// TIA Portal V20 export
// export: Created 2026-08-08T00:00:00.0000000Z, ExportSetting WithDefaults, DisplayName Totally Integrated Automation Portal, DisplayVersion V20, DisplayName TIA Portal Openness, DisplayVersion V20, DisplayName TIA Portal Version Control Interface, DisplayVersion V20, DisplayName STEP 7 Professional, DisplayVersion V20, DisplayName STEP 7 Safety, DisplayVersion V20, DisplayName WinCC Basic/Comfort/Advanced, DisplayVersion V20, DisplayName WinCC Professional, DisplayVersion V20, DisplayName WinCC Unified, DisplayVersion V20
FUNCTION "FC_PhysicalIoCopy" : Void   // FC, SCL
{ S7_Optimized_Access := 'TRUE' }
VERSION : 0.1
// NOT YET WIRED INTO Main[OB1]. Generated 2026-08-08 from the real addresses confirmed live in TIA's Device overview after assigning all 3 ET200SP stations (AFT/MID/FWD) to PLC_1's PROFINET IO system - before that, every module showed no address at all. This is the only block in the whole project that references real physical %I/%Q addresses; everything downstream (FC_IoMapper, Valve_Channels_DB) only ever deals with the abstract 1..368 / 1..208 channel numbers in IO_Buffer_DB. Still needs: (1) FB_ValveLoop simulation guard for real-mapped valves, (2) both this and FC_IoMapper actually called from Main[OB1] - see FC_IoMapper's own header comment. Safe to have present unwired: it only touches IO_Buffer_DB, which nothing else reads yet.
// stored: AutoNumber true, IsIECCheckEnabled false, SetENOAutomatically false, UDAEnableTagReadback false
BEGIN
// Network 1

       // === DIGITAL INPUTS: real %I bits -> IO_Buffer_DB.DI[1..368] ===
       // -- AFT DI modules --
       "IO_Buffer_DB".DI[1] := %I2.0;
       "IO_Buffer_DB".DI[2] := %I2.1;
       "IO_Buffer_DB".DI[3] := %I2.2;
       "IO_Buffer_DB".DI[4] := %I2.3;
       "IO_Buffer_DB".DI[5] := %I2.4;
       "IO_Buffer_DB".DI[6] := %I2.5;
       "IO_Buffer_DB".DI[7] := %I2.6;
       "IO_Buffer_DB".DI[8] := %I2.7;
       "IO_Buffer_DB".DI[9] := %I3.0;
       "IO_Buffer_DB".DI[10] := %I3.1;
       "IO_Buffer_DB".DI[11] := %I3.2;
       "IO_Buffer_DB".DI[12] := %I3.3;
       "IO_Buffer_DB".DI[13] := %I3.4;
       "IO_Buffer_DB".DI[14] := %I3.5;
       "IO_Buffer_DB".DI[15] := %I3.6;
       "IO_Buffer_DB".DI[16] := %I3.7;
       "IO_Buffer_DB".DI[17] := %I4.0;
       "IO_Buffer_DB".DI[18] := %I4.1;
       "IO_Buffer_DB".DI[19] := %I4.2;
       "IO_Buffer_DB".DI[20] := %I4.3;
       "IO_Buffer_DB".DI[21] := %I4.4;
       "IO_Buffer_DB".DI[22] := %I4.5;
       "IO_Buffer_DB".DI[23] := %I4.6;
       "IO_Buffer_DB".DI[24] := %I4.7;
       "IO_Buffer_DB".DI[25] := %I5.0;
       "IO_Buffer_DB".DI[26] := %I5.1;
       "IO_Buffer_DB".DI[27] := %I5.2;
       "IO_Buffer_DB".DI[28] := %I5.3;
       "IO_Buffer_DB".DI[29] := %I5.4;
       "IO_Buffer_DB".DI[30] := %I5.5;
       "IO_Buffer_DB".DI[31] := %I5.6;
       "IO_Buffer_DB".DI[32] := %I5.7;
       "IO_Buffer_DB".DI[33] := %I6.0;
       "IO_Buffer_DB".DI[34] := %I6.1;
       "IO_Buffer_DB".DI[35] := %I6.2;
       "IO_Buffer_DB".DI[36] := %I6.3;
       "IO_Buffer_DB".DI[37] := %I6.4;
       "IO_Buffer_DB".DI[38] := %I6.5;
       "IO_Buffer_DB".DI[39] := %I6.6;
       "IO_Buffer_DB".DI[40] := %I6.7;
       "IO_Buffer_DB".DI[41] := %I7.0;
       "IO_Buffer_DB".DI[42] := %I7.1;
       "IO_Buffer_DB".DI[43] := %I7.2;
       "IO_Buffer_DB".DI[44] := %I7.3;
       "IO_Buffer_DB".DI[45] := %I7.4;
       "IO_Buffer_DB".DI[46] := %I7.5;
       "IO_Buffer_DB".DI[47] := %I7.6;
       "IO_Buffer_DB".DI[48] := %I7.7;
       "IO_Buffer_DB".DI[49] := %I8.0;
       "IO_Buffer_DB".DI[50] := %I8.1;
       "IO_Buffer_DB".DI[51] := %I8.2;
       "IO_Buffer_DB".DI[52] := %I8.3;
       "IO_Buffer_DB".DI[53] := %I8.4;
       "IO_Buffer_DB".DI[54] := %I8.5;
       "IO_Buffer_DB".DI[55] := %I8.6;
       "IO_Buffer_DB".DI[56] := %I8.7;
       "IO_Buffer_DB".DI[57] := %I9.0;
       "IO_Buffer_DB".DI[58] := %I9.1;
       "IO_Buffer_DB".DI[59] := %I9.2;
       "IO_Buffer_DB".DI[60] := %I9.3;
       "IO_Buffer_DB".DI[61] := %I9.4;
       "IO_Buffer_DB".DI[62] := %I9.5;
       "IO_Buffer_DB".DI[63] := %I9.6;
       "IO_Buffer_DB".DI[64] := %I9.7;
       "IO_Buffer_DB".DI[65] := %I10.0;
       "IO_Buffer_DB".DI[66] := %I10.1;
       "IO_Buffer_DB".DI[67] := %I10.2;
       "IO_Buffer_DB".DI[68] := %I10.3;
       "IO_Buffer_DB".DI[69] := %I10.4;
       "IO_Buffer_DB".DI[70] := %I10.5;
       "IO_Buffer_DB".DI[71] := %I10.6;
       "IO_Buffer_DB".DI[72] := %I10.7;
       "IO_Buffer_DB".DI[73] := %I11.0;
       "IO_Buffer_DB".DI[74] := %I11.1;
       "IO_Buffer_DB".DI[75] := %I11.2;
       "IO_Buffer_DB".DI[76] := %I11.3;
       "IO_Buffer_DB".DI[77] := %I11.4;
       "IO_Buffer_DB".DI[78] := %I11.5;
       "IO_Buffer_DB".DI[79] := %I11.6;
       "IO_Buffer_DB".DI[80] := %I11.7;
       "IO_Buffer_DB".DI[81] := %I12.0;
       "IO_Buffer_DB".DI[82] := %I12.1;
       "IO_Buffer_DB".DI[83] := %I12.2;
       "IO_Buffer_DB".DI[84] := %I12.3;
       "IO_Buffer_DB".DI[85] := %I12.4;
       "IO_Buffer_DB".DI[86] := %I12.5;
       "IO_Buffer_DB".DI[87] := %I12.6;
       "IO_Buffer_DB".DI[88] := %I12.7;
       "IO_Buffer_DB".DI[89] := %I13.0;
       "IO_Buffer_DB".DI[90] := %I13.1;
       "IO_Buffer_DB".DI[91] := %I13.2;
       "IO_Buffer_DB".DI[92] := %I13.3;
       "IO_Buffer_DB".DI[93] := %I13.4;
       "IO_Buffer_DB".DI[94] := %I13.5;
       "IO_Buffer_DB".DI[95] := %I13.6;
       "IO_Buffer_DB".DI[96] := %I13.7;
       "IO_Buffer_DB".DI[97] := %I14.0;
       "IO_Buffer_DB".DI[98] := %I14.1;
       "IO_Buffer_DB".DI[99] := %I14.2;
       "IO_Buffer_DB".DI[100] := %I14.3;
       "IO_Buffer_DB".DI[101] := %I14.4;
       "IO_Buffer_DB".DI[102] := %I14.5;
       "IO_Buffer_DB".DI[103] := %I14.6;
       "IO_Buffer_DB".DI[104] := %I14.7;
       "IO_Buffer_DB".DI[105] := %I15.0;
       "IO_Buffer_DB".DI[106] := %I15.1;
       "IO_Buffer_DB".DI[107] := %I15.2;
       "IO_Buffer_DB".DI[108] := %I15.3;
       "IO_Buffer_DB".DI[109] := %I15.4;
       "IO_Buffer_DB".DI[110] := %I15.5;
       "IO_Buffer_DB".DI[111] := %I15.6;
       "IO_Buffer_DB".DI[112] := %I15.7;
       // -- MID DI modules --
       "IO_Buffer_DB".DI[113] := %I16.0;
       "IO_Buffer_DB".DI[114] := %I16.1;
       "IO_Buffer_DB".DI[115] := %I16.2;
       "IO_Buffer_DB".DI[116] := %I16.3;
       "IO_Buffer_DB".DI[117] := %I16.4;
       "IO_Buffer_DB".DI[118] := %I16.5;
       "IO_Buffer_DB".DI[119] := %I16.6;
       "IO_Buffer_DB".DI[120] := %I16.7;
       "IO_Buffer_DB".DI[121] := %I17.0;
       "IO_Buffer_DB".DI[122] := %I17.1;
       "IO_Buffer_DB".DI[123] := %I17.2;
       "IO_Buffer_DB".DI[124] := %I17.3;
       "IO_Buffer_DB".DI[125] := %I17.4;
       "IO_Buffer_DB".DI[126] := %I17.5;
       "IO_Buffer_DB".DI[127] := %I17.6;
       "IO_Buffer_DB".DI[128] := %I17.7;
       "IO_Buffer_DB".DI[129] := %I18.0;
       "IO_Buffer_DB".DI[130] := %I18.1;
       "IO_Buffer_DB".DI[131] := %I18.2;
       "IO_Buffer_DB".DI[132] := %I18.3;
       "IO_Buffer_DB".DI[133] := %I18.4;
       "IO_Buffer_DB".DI[134] := %I18.5;
       "IO_Buffer_DB".DI[135] := %I18.6;
       "IO_Buffer_DB".DI[136] := %I18.7;
       "IO_Buffer_DB".DI[137] := %I19.0;
       "IO_Buffer_DB".DI[138] := %I19.1;
       "IO_Buffer_DB".DI[139] := %I19.2;
       "IO_Buffer_DB".DI[140] := %I19.3;
       "IO_Buffer_DB".DI[141] := %I19.4;
       "IO_Buffer_DB".DI[142] := %I19.5;
       "IO_Buffer_DB".DI[143] := %I19.6;
       "IO_Buffer_DB".DI[144] := %I19.7;
       "IO_Buffer_DB".DI[145] := %I20.0;
       "IO_Buffer_DB".DI[146] := %I20.1;
       "IO_Buffer_DB".DI[147] := %I20.2;
       "IO_Buffer_DB".DI[148] := %I20.3;
       "IO_Buffer_DB".DI[149] := %I20.4;
       "IO_Buffer_DB".DI[150] := %I20.5;
       "IO_Buffer_DB".DI[151] := %I20.6;
       "IO_Buffer_DB".DI[152] := %I20.7;
       "IO_Buffer_DB".DI[153] := %I21.0;
       "IO_Buffer_DB".DI[154] := %I21.1;
       "IO_Buffer_DB".DI[155] := %I21.2;
       "IO_Buffer_DB".DI[156] := %I21.3;
       "IO_Buffer_DB".DI[157] := %I21.4;
       "IO_Buffer_DB".DI[158] := %I21.5;
       "IO_Buffer_DB".DI[159] := %I21.6;
       "IO_Buffer_DB".DI[160] := %I21.7;
       "IO_Buffer_DB".DI[161] := %I22.0;
       "IO_Buffer_DB".DI[162] := %I22.1;
       "IO_Buffer_DB".DI[163] := %I22.2;
       "IO_Buffer_DB".DI[164] := %I22.3;
       "IO_Buffer_DB".DI[165] := %I22.4;
       "IO_Buffer_DB".DI[166] := %I22.5;
       "IO_Buffer_DB".DI[167] := %I22.6;
       "IO_Buffer_DB".DI[168] := %I22.7;
       "IO_Buffer_DB".DI[169] := %I23.0;
       "IO_Buffer_DB".DI[170] := %I23.1;
       "IO_Buffer_DB".DI[171] := %I23.2;
       "IO_Buffer_DB".DI[172] := %I23.3;
       "IO_Buffer_DB".DI[173] := %I23.4;
       "IO_Buffer_DB".DI[174] := %I23.5;
       "IO_Buffer_DB".DI[175] := %I23.6;
       "IO_Buffer_DB".DI[176] := %I23.7;
       "IO_Buffer_DB".DI[177] := %I24.0;
       "IO_Buffer_DB".DI[178] := %I24.1;
       "IO_Buffer_DB".DI[179] := %I24.2;
       "IO_Buffer_DB".DI[180] := %I24.3;
       "IO_Buffer_DB".DI[181] := %I24.4;
       "IO_Buffer_DB".DI[182] := %I24.5;
       "IO_Buffer_DB".DI[183] := %I24.6;
       "IO_Buffer_DB".DI[184] := %I24.7;
       "IO_Buffer_DB".DI[185] := %I25.0;
       "IO_Buffer_DB".DI[186] := %I25.1;
       "IO_Buffer_DB".DI[187] := %I25.2;
       "IO_Buffer_DB".DI[188] := %I25.3;
       "IO_Buffer_DB".DI[189] := %I25.4;
       "IO_Buffer_DB".DI[190] := %I25.5;
       "IO_Buffer_DB".DI[191] := %I25.6;
       "IO_Buffer_DB".DI[192] := %I25.7;
       "IO_Buffer_DB".DI[193] := %I26.0;
       "IO_Buffer_DB".DI[194] := %I26.1;
       "IO_Buffer_DB".DI[195] := %I26.2;
       "IO_Buffer_DB".DI[196] := %I26.3;
       "IO_Buffer_DB".DI[197] := %I26.4;
       "IO_Buffer_DB".DI[198] := %I26.5;
       "IO_Buffer_DB".DI[199] := %I26.6;
       "IO_Buffer_DB".DI[200] := %I26.7;
       "IO_Buffer_DB".DI[201] := %I27.0;
       "IO_Buffer_DB".DI[202] := %I27.1;
       "IO_Buffer_DB".DI[203] := %I27.2;
       "IO_Buffer_DB".DI[204] := %I27.3;
       "IO_Buffer_DB".DI[205] := %I27.4;
       "IO_Buffer_DB".DI[206] := %I27.5;
       "IO_Buffer_DB".DI[207] := %I27.6;
       "IO_Buffer_DB".DI[208] := %I27.7;
       "IO_Buffer_DB".DI[209] := %I28.0;
       "IO_Buffer_DB".DI[210] := %I28.1;
       "IO_Buffer_DB".DI[211] := %I28.2;
       "IO_Buffer_DB".DI[212] := %I28.3;
       "IO_Buffer_DB".DI[213] := %I28.4;
       "IO_Buffer_DB".DI[214] := %I28.5;
       "IO_Buffer_DB".DI[215] := %I28.6;
       "IO_Buffer_DB".DI[216] := %I28.7;
       "IO_Buffer_DB".DI[217] := %I29.0;
       "IO_Buffer_DB".DI[218] := %I29.1;
       "IO_Buffer_DB".DI[219] := %I29.2;
       "IO_Buffer_DB".DI[220] := %I29.3;
       "IO_Buffer_DB".DI[221] := %I29.4;
       "IO_Buffer_DB".DI[222] := %I29.5;
       "IO_Buffer_DB".DI[223] := %I29.6;
       "IO_Buffer_DB".DI[224] := %I29.7;
       // -- FWD DI modules --
       "IO_Buffer_DB".DI[225] := %I30.0;
       "IO_Buffer_DB".DI[226] := %I30.1;
       "IO_Buffer_DB".DI[227] := %I30.2;
       "IO_Buffer_DB".DI[228] := %I30.3;
       "IO_Buffer_DB".DI[229] := %I30.4;
       "IO_Buffer_DB".DI[230] := %I30.5;
       "IO_Buffer_DB".DI[231] := %I30.6;
       "IO_Buffer_DB".DI[232] := %I30.7;
       "IO_Buffer_DB".DI[233] := %I31.0;
       "IO_Buffer_DB".DI[234] := %I31.1;
       "IO_Buffer_DB".DI[235] := %I31.2;
       "IO_Buffer_DB".DI[236] := %I31.3;
       "IO_Buffer_DB".DI[237] := %I31.4;
       "IO_Buffer_DB".DI[238] := %I31.5;
       "IO_Buffer_DB".DI[239] := %I31.6;
       "IO_Buffer_DB".DI[240] := %I31.7;
       "IO_Buffer_DB".DI[241] := %I32.0;
       "IO_Buffer_DB".DI[242] := %I32.1;
       "IO_Buffer_DB".DI[243] := %I32.2;
       "IO_Buffer_DB".DI[244] := %I32.3;
       "IO_Buffer_DB".DI[245] := %I32.4;
       "IO_Buffer_DB".DI[246] := %I32.5;
       "IO_Buffer_DB".DI[247] := %I32.6;
       "IO_Buffer_DB".DI[248] := %I32.7;
       "IO_Buffer_DB".DI[249] := %I33.0;
       "IO_Buffer_DB".DI[250] := %I33.1;
       "IO_Buffer_DB".DI[251] := %I33.2;
       "IO_Buffer_DB".DI[252] := %I33.3;
       "IO_Buffer_DB".DI[253] := %I33.4;
       "IO_Buffer_DB".DI[254] := %I33.5;
       "IO_Buffer_DB".DI[255] := %I33.6;
       "IO_Buffer_DB".DI[256] := %I33.7;
       "IO_Buffer_DB".DI[257] := %I34.0;
       "IO_Buffer_DB".DI[258] := %I34.1;
       "IO_Buffer_DB".DI[259] := %I34.2;
       "IO_Buffer_DB".DI[260] := %I34.3;
       "IO_Buffer_DB".DI[261] := %I34.4;
       "IO_Buffer_DB".DI[262] := %I34.5;
       "IO_Buffer_DB".DI[263] := %I34.6;
       "IO_Buffer_DB".DI[264] := %I34.7;
       "IO_Buffer_DB".DI[265] := %I35.0;
       "IO_Buffer_DB".DI[266] := %I35.1;
       "IO_Buffer_DB".DI[267] := %I35.2;
       "IO_Buffer_DB".DI[268] := %I35.3;
       "IO_Buffer_DB".DI[269] := %I35.4;
       "IO_Buffer_DB".DI[270] := %I35.5;
       "IO_Buffer_DB".DI[271] := %I35.6;
       "IO_Buffer_DB".DI[272] := %I35.7;
       "IO_Buffer_DB".DI[273] := %I36.0;
       "IO_Buffer_DB".DI[274] := %I36.1;
       "IO_Buffer_DB".DI[275] := %I36.2;
       "IO_Buffer_DB".DI[276] := %I36.3;
       "IO_Buffer_DB".DI[277] := %I36.4;
       "IO_Buffer_DB".DI[278] := %I36.5;
       "IO_Buffer_DB".DI[279] := %I36.6;
       "IO_Buffer_DB".DI[280] := %I36.7;
       "IO_Buffer_DB".DI[281] := %I37.0;
       "IO_Buffer_DB".DI[282] := %I37.1;
       "IO_Buffer_DB".DI[283] := %I37.2;
       "IO_Buffer_DB".DI[284] := %I37.3;
       "IO_Buffer_DB".DI[285] := %I37.4;
       "IO_Buffer_DB".DI[286] := %I37.5;
       "IO_Buffer_DB".DI[287] := %I37.6;
       "IO_Buffer_DB".DI[288] := %I37.7;
       "IO_Buffer_DB".DI[289] := %I38.0;
       "IO_Buffer_DB".DI[290] := %I38.1;
       "IO_Buffer_DB".DI[291] := %I38.2;
       "IO_Buffer_DB".DI[292] := %I38.3;
       "IO_Buffer_DB".DI[293] := %I38.4;
       "IO_Buffer_DB".DI[294] := %I38.5;
       "IO_Buffer_DB".DI[295] := %I38.6;
       "IO_Buffer_DB".DI[296] := %I38.7;
       "IO_Buffer_DB".DI[297] := %I39.0;
       "IO_Buffer_DB".DI[298] := %I39.1;
       "IO_Buffer_DB".DI[299] := %I39.2;
       "IO_Buffer_DB".DI[300] := %I39.3;
       "IO_Buffer_DB".DI[301] := %I39.4;
       "IO_Buffer_DB".DI[302] := %I39.5;
       "IO_Buffer_DB".DI[303] := %I39.6;
       "IO_Buffer_DB".DI[304] := %I39.7;
       "IO_Buffer_DB".DI[305] := %I40.0;
       "IO_Buffer_DB".DI[306] := %I40.1;
       "IO_Buffer_DB".DI[307] := %I40.2;
       "IO_Buffer_DB".DI[308] := %I40.3;
       "IO_Buffer_DB".DI[309] := %I40.4;
       "IO_Buffer_DB".DI[310] := %I40.5;
       "IO_Buffer_DB".DI[311] := %I40.6;
       "IO_Buffer_DB".DI[312] := %I40.7;
       "IO_Buffer_DB".DI[313] := %I41.0;
       "IO_Buffer_DB".DI[314] := %I41.1;
       "IO_Buffer_DB".DI[315] := %I41.2;
       "IO_Buffer_DB".DI[316] := %I41.3;
       "IO_Buffer_DB".DI[317] := %I41.4;
       "IO_Buffer_DB".DI[318] := %I41.5;
       "IO_Buffer_DB".DI[319] := %I41.6;
       "IO_Buffer_DB".DI[320] := %I41.7;
       "IO_Buffer_DB".DI[321] := %I42.0;
       "IO_Buffer_DB".DI[322] := %I42.1;
       "IO_Buffer_DB".DI[323] := %I42.2;
       "IO_Buffer_DB".DI[324] := %I42.3;
       "IO_Buffer_DB".DI[325] := %I42.4;
       "IO_Buffer_DB".DI[326] := %I42.5;
       "IO_Buffer_DB".DI[327] := %I42.6;
       "IO_Buffer_DB".DI[328] := %I42.7;
       "IO_Buffer_DB".DI[329] := %I43.0;
       "IO_Buffer_DB".DI[330] := %I43.1;
       "IO_Buffer_DB".DI[331] := %I43.2;
       "IO_Buffer_DB".DI[332] := %I43.3;
       "IO_Buffer_DB".DI[333] := %I43.4;
       "IO_Buffer_DB".DI[334] := %I43.5;
       "IO_Buffer_DB".DI[335] := %I43.6;
       "IO_Buffer_DB".DI[336] := %I43.7;
       "IO_Buffer_DB".DI[337] := %I44.0;
       "IO_Buffer_DB".DI[338] := %I44.1;
       "IO_Buffer_DB".DI[339] := %I44.2;
       "IO_Buffer_DB".DI[340] := %I44.3;
       "IO_Buffer_DB".DI[341] := %I44.4;
       "IO_Buffer_DB".DI[342] := %I44.5;
       "IO_Buffer_DB".DI[343] := %I44.6;
       "IO_Buffer_DB".DI[344] := %I44.7;
       "IO_Buffer_DB".DI[345] := %I45.0;
       "IO_Buffer_DB".DI[346] := %I45.1;
       "IO_Buffer_DB".DI[347] := %I45.2;
       "IO_Buffer_DB".DI[348] := %I45.3;
       "IO_Buffer_DB".DI[349] := %I45.4;
       "IO_Buffer_DB".DI[350] := %I45.5;
       "IO_Buffer_DB".DI[351] := %I45.6;
       "IO_Buffer_DB".DI[352] := %I45.7;
       "IO_Buffer_DB".DI[353] := %I46.0;
       "IO_Buffer_DB".DI[354] := %I46.1;
       "IO_Buffer_DB".DI[355] := %I46.2;
       "IO_Buffer_DB".DI[356] := %I46.3;
       "IO_Buffer_DB".DI[357] := %I46.4;
       "IO_Buffer_DB".DI[358] := %I46.5;
       "IO_Buffer_DB".DI[359] := %I46.6;
       "IO_Buffer_DB".DI[360] := %I46.7;
       "IO_Buffer_DB".DI[361] := %I47.0;
       "IO_Buffer_DB".DI[362] := %I47.1;
       "IO_Buffer_DB".DI[363] := %I47.2;
       "IO_Buffer_DB".DI[364] := %I47.3;
       "IO_Buffer_DB".DI[365] := %I47.4;
       "IO_Buffer_DB".DI[366] := %I47.5;
       "IO_Buffer_DB".DI[367] := %I47.6;
       "IO_Buffer_DB".DI[368] := %I47.7;

       // === DIGITAL OUTPUTS: IO_Buffer_DB.DQ[1..208] -> real %Q bits ===
       // -- AFT DQ modules --
       %Q2.0 := "IO_Buffer_DB".DQ[1];
       %Q2.1 := "IO_Buffer_DB".DQ[2];
       %Q2.2 := "IO_Buffer_DB".DQ[3];
       %Q2.3 := "IO_Buffer_DB".DQ[4];
       %Q2.4 := "IO_Buffer_DB".DQ[5];
       %Q2.5 := "IO_Buffer_DB".DQ[6];
       %Q2.6 := "IO_Buffer_DB".DQ[7];
       %Q2.7 := "IO_Buffer_DB".DQ[8];
       %Q3.0 := "IO_Buffer_DB".DQ[9];
       %Q3.1 := "IO_Buffer_DB".DQ[10];
       %Q3.2 := "IO_Buffer_DB".DQ[11];
       %Q3.3 := "IO_Buffer_DB".DQ[12];
       %Q3.4 := "IO_Buffer_DB".DQ[13];
       %Q3.5 := "IO_Buffer_DB".DQ[14];
       %Q3.6 := "IO_Buffer_DB".DQ[15];
       %Q3.7 := "IO_Buffer_DB".DQ[16];
       %Q4.0 := "IO_Buffer_DB".DQ[17];
       %Q4.1 := "IO_Buffer_DB".DQ[18];
       %Q4.2 := "IO_Buffer_DB".DQ[19];
       %Q4.3 := "IO_Buffer_DB".DQ[20];
       %Q4.4 := "IO_Buffer_DB".DQ[21];
       %Q4.5 := "IO_Buffer_DB".DQ[22];
       %Q4.6 := "IO_Buffer_DB".DQ[23];
       %Q4.7 := "IO_Buffer_DB".DQ[24];
       %Q5.0 := "IO_Buffer_DB".DQ[25];
       %Q5.1 := "IO_Buffer_DB".DQ[26];
       %Q5.2 := "IO_Buffer_DB".DQ[27];
       %Q5.3 := "IO_Buffer_DB".DQ[28];
       %Q5.4 := "IO_Buffer_DB".DQ[29];
       %Q5.5 := "IO_Buffer_DB".DQ[30];
       %Q5.6 := "IO_Buffer_DB".DQ[31];
       %Q5.7 := "IO_Buffer_DB".DQ[32];
       %Q6.0 := "IO_Buffer_DB".DQ[33];
       %Q6.1 := "IO_Buffer_DB".DQ[34];
       %Q6.2 := "IO_Buffer_DB".DQ[35];
       %Q6.3 := "IO_Buffer_DB".DQ[36];
       %Q6.4 := "IO_Buffer_DB".DQ[37];
       %Q6.5 := "IO_Buffer_DB".DQ[38];
       %Q6.6 := "IO_Buffer_DB".DQ[39];
       %Q6.7 := "IO_Buffer_DB".DQ[40];
       %Q7.0 := "IO_Buffer_DB".DQ[41];
       %Q7.1 := "IO_Buffer_DB".DQ[42];
       %Q7.2 := "IO_Buffer_DB".DQ[43];
       %Q7.3 := "IO_Buffer_DB".DQ[44];
       %Q7.4 := "IO_Buffer_DB".DQ[45];
       %Q7.5 := "IO_Buffer_DB".DQ[46];
       %Q7.6 := "IO_Buffer_DB".DQ[47];
       %Q7.7 := "IO_Buffer_DB".DQ[48];
       %Q8.0 := "IO_Buffer_DB".DQ[49];
       %Q8.1 := "IO_Buffer_DB".DQ[50];
       %Q8.2 := "IO_Buffer_DB".DQ[51];
       %Q8.3 := "IO_Buffer_DB".DQ[52];
       %Q8.4 := "IO_Buffer_DB".DQ[53];
       %Q8.5 := "IO_Buffer_DB".DQ[54];
       %Q8.6 := "IO_Buffer_DB".DQ[55];
       %Q8.7 := "IO_Buffer_DB".DQ[56];
       %Q9.0 := "IO_Buffer_DB".DQ[57];
       %Q9.1 := "IO_Buffer_DB".DQ[58];
       %Q9.2 := "IO_Buffer_DB".DQ[59];
       %Q9.3 := "IO_Buffer_DB".DQ[60];
       %Q9.4 := "IO_Buffer_DB".DQ[61];
       %Q9.5 := "IO_Buffer_DB".DQ[62];
       %Q9.6 := "IO_Buffer_DB".DQ[63];
       %Q9.7 := "IO_Buffer_DB".DQ[64];
       // -- MID DQ modules --
       %Q10.0 := "IO_Buffer_DB".DQ[65];
       %Q10.1 := "IO_Buffer_DB".DQ[66];
       %Q10.2 := "IO_Buffer_DB".DQ[67];
       %Q10.3 := "IO_Buffer_DB".DQ[68];
       %Q10.4 := "IO_Buffer_DB".DQ[69];
       %Q10.5 := "IO_Buffer_DB".DQ[70];
       %Q10.6 := "IO_Buffer_DB".DQ[71];
       %Q10.7 := "IO_Buffer_DB".DQ[72];
       %Q11.0 := "IO_Buffer_DB".DQ[73];
       %Q11.1 := "IO_Buffer_DB".DQ[74];
       %Q11.2 := "IO_Buffer_DB".DQ[75];
       %Q11.3 := "IO_Buffer_DB".DQ[76];
       %Q11.4 := "IO_Buffer_DB".DQ[77];
       %Q11.5 := "IO_Buffer_DB".DQ[78];
       %Q11.6 := "IO_Buffer_DB".DQ[79];
       %Q11.7 := "IO_Buffer_DB".DQ[80];
       %Q12.0 := "IO_Buffer_DB".DQ[81];
       %Q12.1 := "IO_Buffer_DB".DQ[82];
       %Q12.2 := "IO_Buffer_DB".DQ[83];
       %Q12.3 := "IO_Buffer_DB".DQ[84];
       %Q12.4 := "IO_Buffer_DB".DQ[85];
       %Q12.5 := "IO_Buffer_DB".DQ[86];
       %Q12.6 := "IO_Buffer_DB".DQ[87];
       %Q12.7 := "IO_Buffer_DB".DQ[88];
       %Q13.0 := "IO_Buffer_DB".DQ[89];
       %Q13.1 := "IO_Buffer_DB".DQ[90];
       %Q13.2 := "IO_Buffer_DB".DQ[91];
       %Q13.3 := "IO_Buffer_DB".DQ[92];
       %Q13.4 := "IO_Buffer_DB".DQ[93];
       %Q13.5 := "IO_Buffer_DB".DQ[94];
       %Q13.6 := "IO_Buffer_DB".DQ[95];
       %Q13.7 := "IO_Buffer_DB".DQ[96];
       %Q14.0 := "IO_Buffer_DB".DQ[97];
       %Q14.1 := "IO_Buffer_DB".DQ[98];
       %Q14.2 := "IO_Buffer_DB".DQ[99];
       %Q14.3 := "IO_Buffer_DB".DQ[100];
       %Q14.4 := "IO_Buffer_DB".DQ[101];
       %Q14.5 := "IO_Buffer_DB".DQ[102];
       %Q14.6 := "IO_Buffer_DB".DQ[103];
       %Q14.7 := "IO_Buffer_DB".DQ[104];
       %Q15.0 := "IO_Buffer_DB".DQ[105];
       %Q15.1 := "IO_Buffer_DB".DQ[106];
       %Q15.2 := "IO_Buffer_DB".DQ[107];
       %Q15.3 := "IO_Buffer_DB".DQ[108];
       %Q15.4 := "IO_Buffer_DB".DQ[109];
       %Q15.5 := "IO_Buffer_DB".DQ[110];
       %Q15.6 := "IO_Buffer_DB".DQ[111];
       %Q15.7 := "IO_Buffer_DB".DQ[112];
       %Q16.0 := "IO_Buffer_DB".DQ[113];
       %Q16.1 := "IO_Buffer_DB".DQ[114];
       %Q16.2 := "IO_Buffer_DB".DQ[115];
       %Q16.3 := "IO_Buffer_DB".DQ[116];
       %Q16.4 := "IO_Buffer_DB".DQ[117];
       %Q16.5 := "IO_Buffer_DB".DQ[118];
       %Q16.6 := "IO_Buffer_DB".DQ[119];
       %Q16.7 := "IO_Buffer_DB".DQ[120];
       %Q17.0 := "IO_Buffer_DB".DQ[121];
       %Q17.1 := "IO_Buffer_DB".DQ[122];
       %Q17.2 := "IO_Buffer_DB".DQ[123];
       %Q17.3 := "IO_Buffer_DB".DQ[124];
       %Q17.4 := "IO_Buffer_DB".DQ[125];
       %Q17.5 := "IO_Buffer_DB".DQ[126];
       %Q17.6 := "IO_Buffer_DB".DQ[127];
       %Q17.7 := "IO_Buffer_DB".DQ[128];
       // -- FWD DQ modules --
       %Q18.0 := "IO_Buffer_DB".DQ[129];
       %Q18.1 := "IO_Buffer_DB".DQ[130];
       %Q18.2 := "IO_Buffer_DB".DQ[131];
       %Q18.3 := "IO_Buffer_DB".DQ[132];
       %Q18.4 := "IO_Buffer_DB".DQ[133];
       %Q18.5 := "IO_Buffer_DB".DQ[134];
       %Q18.6 := "IO_Buffer_DB".DQ[135];
       %Q18.7 := "IO_Buffer_DB".DQ[136];
       %Q19.0 := "IO_Buffer_DB".DQ[137];
       %Q19.1 := "IO_Buffer_DB".DQ[138];
       %Q19.2 := "IO_Buffer_DB".DQ[139];
       %Q19.3 := "IO_Buffer_DB".DQ[140];
       %Q19.4 := "IO_Buffer_DB".DQ[141];
       %Q19.5 := "IO_Buffer_DB".DQ[142];
       %Q19.6 := "IO_Buffer_DB".DQ[143];
       %Q19.7 := "IO_Buffer_DB".DQ[144];
       %Q20.0 := "IO_Buffer_DB".DQ[145];
       %Q20.1 := "IO_Buffer_DB".DQ[146];
       %Q20.2 := "IO_Buffer_DB".DQ[147];
       %Q20.3 := "IO_Buffer_DB".DQ[148];
       %Q20.4 := "IO_Buffer_DB".DQ[149];
       %Q20.5 := "IO_Buffer_DB".DQ[150];
       %Q20.6 := "IO_Buffer_DB".DQ[151];
       %Q20.7 := "IO_Buffer_DB".DQ[152];
       %Q21.0 := "IO_Buffer_DB".DQ[153];
       %Q21.1 := "IO_Buffer_DB".DQ[154];
       %Q21.2 := "IO_Buffer_DB".DQ[155];
       %Q21.3 := "IO_Buffer_DB".DQ[156];
       %Q21.4 := "IO_Buffer_DB".DQ[157];
       %Q21.5 := "IO_Buffer_DB".DQ[158];
       %Q21.6 := "IO_Buffer_DB".DQ[159];
       %Q21.7 := "IO_Buffer_DB".DQ[160];
       %Q22.0 := "IO_Buffer_DB".DQ[161];
       %Q22.1 := "IO_Buffer_DB".DQ[162];
       %Q22.2 := "IO_Buffer_DB".DQ[163];
       %Q22.3 := "IO_Buffer_DB".DQ[164];
       %Q22.4 := "IO_Buffer_DB".DQ[165];
       %Q22.5 := "IO_Buffer_DB".DQ[166];
       %Q22.6 := "IO_Buffer_DB".DQ[167];
       %Q22.7 := "IO_Buffer_DB".DQ[168];
       %Q23.0 := "IO_Buffer_DB".DQ[169];
       %Q23.1 := "IO_Buffer_DB".DQ[170];
       %Q23.2 := "IO_Buffer_DB".DQ[171];
       %Q23.3 := "IO_Buffer_DB".DQ[172];
       %Q23.4 := "IO_Buffer_DB".DQ[173];
       %Q23.5 := "IO_Buffer_DB".DQ[174];
       %Q23.6 := "IO_Buffer_DB".DQ[175];
       %Q23.7 := "IO_Buffer_DB".DQ[176];
       %Q24.0 := "IO_Buffer_DB".DQ[177];
       %Q24.1 := "IO_Buffer_DB".DQ[178];
       %Q24.2 := "IO_Buffer_DB".DQ[179];
       %Q24.3 := "IO_Buffer_DB".DQ[180];
       %Q24.4 := "IO_Buffer_DB".DQ[181];
       %Q24.5 := "IO_Buffer_DB".DQ[182];
       %Q24.6 := "IO_Buffer_DB".DQ[183];
       %Q24.7 := "IO_Buffer_DB".DQ[184];
       %Q25.0 := "IO_Buffer_DB".DQ[185];
       %Q25.1 := "IO_Buffer_DB".DQ[186];
       %Q25.2 := "IO_Buffer_DB".DQ[187];
       %Q25.3 := "IO_Buffer_DB".DQ[188];
       %Q25.4 := "IO_Buffer_DB".DQ[189];
       %Q25.5 := "IO_Buffer_DB".DQ[190];
       %Q25.6 := "IO_Buffer_DB".DQ[191];
       %Q25.7 := "IO_Buffer_DB".DQ[192];
       %Q26.0 := "IO_Buffer_DB".DQ[193];
       %Q26.1 := "IO_Buffer_DB".DQ[194];
       %Q26.2 := "IO_Buffer_DB".DQ[195];
       %Q26.3 := "IO_Buffer_DB".DQ[196];
       %Q26.4 := "IO_Buffer_DB".DQ[197];
       %Q26.5 := "IO_Buffer_DB".DQ[198];
       %Q26.6 := "IO_Buffer_DB".DQ[199];
       %Q26.7 := "IO_Buffer_DB".DQ[200];
       %Q27.0 := "IO_Buffer_DB".DQ[201];
       %Q27.1 := "IO_Buffer_DB".DQ[202];
       %Q27.2 := "IO_Buffer_DB".DQ[203];
       %Q27.3 := "IO_Buffer_DB".DQ[204];
       %Q27.4 := "IO_Buffer_DB".DQ[205];
       %Q27.5 := "IO_Buffer_DB".DQ[206];
       %Q27.6 := "IO_Buffer_DB".DQ[207];
       %Q27.7 := "IO_Buffer_DB".DQ[208];
END_FUNCTION
